Staubli VAL3: jointSpace.dtx

public jointRx jJointPos
public JointVel jJointVel
  [0]
    num jv1
    num jv2
    num jv3
    num jv4
    num jv5
    num jv6
public JointAccel jJointAccel
  [0]
    num ja1
    num ja2
    num ja3
    num ja4
    num ja5
    num ja6
public JointForce jJointForce
  [0]
    num jf1
    num jf2
    num jf3
    num jf4
    num jf5
    num jf6
